// SIMATIC S7-200 project (STEP 7-Micro/WIN), CPU 226 REL 01.00

SYMBOL_TABLE SYM1
                 M0.0     // 0
END_SYMBOL_TABLE

ORGANIZATION_BLOCK OB_1:OB1
TITLE=【S7-200 PLC与DDM4A数显表的通信控制系统（一）】
// 我设计的程序用于实现在工业自动化场景多路温度监测系统，用于实时显示多达 16 个通道的温度值。
// 系统的工作流程如下：主程序块在PLC启动时初始化数据，将脉冲进程标志设置为1，并持续调用显示驱动子程序。在显示驱动子程序中，选通端口通过移位操作生成8组选通信号，依次选择显示通道，其移位操作按顺序执行，避免显示混乱。
// 数据显示方面，16个通道的温度值存储在相应的存储区域中。例如，当某个通道更新控制位为ON时，通道1的温度值增加，但其值保持在0到9999之间，避免溢出。这些数据经过IBCD转换后存储到临时数据存储中。随后，通过位操作分解为千位、百位、十位、个位和小数点数据，其格式与数显表要求一致。
// 在数据输出阶段，例如，某个脉冲进程控制位触发时通过数据输出端口输出个位数据，另一个控制位触发时输出千位数据。这些控制位按顺序触发，确保数显表按序显示每个通道的温度值。
// 
BEGIN
Network 1
LD     SM0.1
MOVB   1, QB1
MOVW   +1, MW1
Network 2
LD     SM0.0
CALL   SBR_0:SBR0
Network 3
LD     Q1.0
EU
INCW   VW50
AW>=   VW50, +9999
MOVW   +0, VW50
Network 4
LD     Q1.1
EU
LPS
INCW   VW54
AW>=   VW54, +9999
MOVW   +0, VW54
LRD
INCW   VW56
LPP
AW>=   VW56, +16
MOVW   +0, VW56
END_ORGANIZATION_BLOCK

SUBROUTINE_BLOCK SBR_0:SBR0
TITLE= 
// SUBROUTINE COMMENTS
// Press F1 for help and example program
//  
BEGIN
Network 1 // 产生16个数据脉冲进程
//  
// NETWORK COMMENTS
//  
// 
LD     T32
EU
RLW    MW1, 1
Network 2 // 产生8组选通
// 
// 
LD     M2.7
EU
RLB    QB1, 1
Network 3 // 产生脉冲，脉冲宽度＝VW2；1单位＝1ms
// 
// 
LDN    T32
TON    T32, VW2
Network 4 // 显示数据1、9（显示数据1~8＝VW50~VW80）（显示数据9~16＝VW82~VW112）
// 
// 
// 
LD     Q1.0
MOVW   VW50, MW10
IBCD   MW10
MOVW   VW52, MW12
IBCD   MW12
MOVW   VW82, MW14
IBCD   MW14
MOVW   VW84, MW16
IBCD   MW16
Network 5 // 显示数据2、10
// 
// 
LD     Q1.1
MOVW   VW54, MW10
IBCD   MW10
MOVW   VW56, MW12
IBCD   MW12
MOVW   VW86, MW14
IBCD   MW14
MOVW   VW88, MW16
IBCD   MW16
Network 6 // 显示数据3、11
// 
// 
LD     Q1.2
MOVW   VW58, MW10
IBCD   MW10
MOVW   VW60, MW12
IBCD   MW12
MOVW   VW90, MW14
IBCD   MW14
MOVW   VW92, MW16
IBCD   MW16
Network 7 // 显示数据4、12
// 
// 
LD     Q1.3
MOVW   VW62, MW10
IBCD   MW10
MOVW   VW64, MW12
IBCD   MW12
MOVW   VW94, MW14
IBCD   MW14
MOVW   VW96, MW16
IBCD   MW16
Network 8 // 显示数据5、13
// 
// 
LD     Q1.4
MOVW   VW66, MW10
IBCD   MW10
MOVW   VW68, MW12
IBCD   MW12
MOVW   VW98, MW14
IBCD   MW14
MOVW   VW100, MW16
IBCD   MW16
Network 9 // 显示数据6、14
// 
// 
LD     Q1.5
MOVW   VW70, MW10
IBCD   MW10
MOVW   VW72, MW12
IBCD   MW12
MOVW   VW102, MW14
IBCD   MW14
MOVW   VW104, MW16
IBCD   MW16
Network 10 // 显示数据7、15
// 
// 
LD     Q1.6
MOVW   VW74, MW10
IBCD   MW10
MOVW   VW76, MW12
IBCD   MW12
MOVW   VW106, MW14
IBCD   MW14
MOVW   VW108, MW16
IBCD   MW16
Network 11 // 显示数据8、16
// 
// 
LD     Q1.7
MOVW   VW78, MW10
IBCD   MW10
MOVW   VW80, MW12
IBCD   MW12
MOVW   VW110, MW14
IBCD   MW14
MOVW   VW112, MW16
IBCD   MW16
Network 12 // 合成千位数据
// 
// 
LD     SM0.0
LPS
MOVB   MB14, LB4
ANDB   240, LB4
MOVB   MB10, LB0
SRB    LB0, 4
AN     Q1.1
MOVB   LB0, LB10
ORB    LB4, LB10
LRD
MOVB   VB57, LB20
LRD
MOVB   LB20, LB21
ANDB   15, LB21
LPP
A      Q1.1
MOVB   LB0, LB10
ORB    LB21, LB10
Network 13 // 合成百位数据
// 
// 
LD     SM0.0
MOVB   MB10, LB1
ANDB   15, LB1
MOVB   MB14, LB5
SLB    LB5, 4
MOVB   LB1, LB11
ORB    LB5, LB11
Network 14 // 合成十位数据
// 
// 
LD     SM0.0
MOVB   MB15, LB6
ANDB   240, LB6
MOVB   MB11, LB2
SRB    LB2, 4
MOVB   LB2, LB12
ORB    LB6, LB12
Network 15 // 合成个位数据
// 
// 
LD     SM0.0
MOVB   MB11, LB3
ANDB   15, LB3
MOVB   MB15, LB7
SLB    LB7, 4
MOVB   LB3, LB13
ORB    LB7, LB13
Network 16 // 合成小数点数据
// 
// 
LD     SM0.0
MOVB   MB13, LB8
ANDB   15, LB8
MOVB   MB17, LB9
SLB    LB9, 4
MOVB   LB8, LB14
ORB    LB9, LB14
Network 17 // 脉冲进程1
// 
// 
LD     M1.0
MOVB   255, QB0
Network 18 // 脉冲进程2
// 
// 
LD     M1.1
MOVB   0, QB0
Network 19 // 脉冲进程3
// 
// 
LD     M1.2
MOVB   238, QB0
Network 20 // 脉冲进程4
// 
// 
LD     M1.3
MOVB   255, QB0
Network 21 // 脉冲进程5
// 
// 
LD     M1.4
MOVB   LB13, QB0
Network 22 // 脉冲进程6
// 
// 
LD     M1.5
MOVB   255, QB0
Network 23 // 脉冲进程7
// 
// 
LD     M1.6
MOVB   LB12, QB0
Network 24 // 脉冲进程8
// 
// 
LD     M1.7
MOVB   255, QB0
Network 25 // 脉冲进程9
// 
// 
LD     M2.0
MOVB   LB11, QB0
Network 26 // 脉冲进程10
// 
// 
LD     M2.1
MOVB   255, QB0
Network 27 // 脉冲进程11
// 
// 
LD     M2.2
MOVB   LB10, QB0
Network 28 // 脉冲进程12
// 
// 
LD     M2.3
MOVB   255, QB0
Network 29 // 脉冲进程13
// 
// 
LD     M2.4
MOVB   LB14, QB0
Network 30 // 脉冲进程14
// 
// 
LD     M2.5
MOVB   255, QB0
Network 31 // 脉冲进程15
// 
// 
LD     M2.6
MOVB   0, QB0
END_SUBROUTINE_BLOCK

INTERRUPT_BLOCK INT_0:INT0
TITLE= 
// INTERRUPT ROUTINE COMMENTS
// Press F1 for help and example program
//  
BEGIN
Network 1
LD     SM0.0
=      M0.0
Network 2 // NETWORK TITLE (single line)
//  
// NETWORK COMMENTS
//  
// 
END_INTERRUPT_BLOCK
